Staubli VAL3: onEdit.pgx

public program onEdit(string& x_sItem[])
  local num l_nX
  local num l_nY
  local num l_nDelay
  local bool l_bValide
  local num l_nIndex
  local num l_nOperator
  local num l_nValue
  local string l_sType
  local string l_sName
begin
  // decompose it
  call saveInOut:decompose_wait(x_sItem,l_sName,l_nOperator,l_nValue)
  if l_sName!=""
    // get the item
    call saveInOut:get_num(x_sItem,l_nIndex)
    // edit it
    call make_it(x_sItem)
  else
    x_sItem=""
  endIf
end
